// TIA Portal V18 export
FUNCTION "Boiler_UnitState" : Void   // FC61000, FBD
{ S7_Optimized_Access := 'TRUE' }
VERSION : 0.1
// BoilerOpMode                                        BoilerUnitState
// 0-OFF/Summer                                       0 Off
// 1-On/Winter                                             1 ColdStandBy
//                                                                   1 HotStandBy
//                                                                   2 Heating
// stored: AutoNumber false, IsIECCheckEnabled false, SetENOAutomatically false, UDAEnableTagReadback false
   VAR_INPUT
      rOAT : Real;
      rBoiler1OATOff : Real;
      rBoiler1OATOn : Real;
      rBoiler2OAT1On : Real;
      rBoiler2OAT1Off : Real;
      rBoiler2OAT2On : Real;
      rBoiler2OAT2Off : Real;
   END_VAR
   VAR_IN_OUT
      xBoiler1OATRequest : Bool;
      xBoiler2OATRequest : Bool;
   END_VAR
   VAR_TEMP
      FA_temp : Real;
      xB1State : Bool;
      xB2Band1State : Bool;
      xB2Band2State : Bool;
      xB2Band1Effective : Bool;
   END_VAR
BEGIN

REGION Network 1 (SCL)
   IF "FirstScan" THEN
       ;
       //"AHUUnitStates".UnitStates.cActual[#iUnitID] := 0;
       //"AHUUnitStates".UnitStates.cTarget[#iUnitID] := 0;
   END_IF;
END_REGION

REGION Network 2 (SCL): Boiler1 Select from Panel
   IF "HSsDI".Requests.xSeasonAuto[1] THEN
       "BoilerOpModes".OpModes.cPreselectedOpModePanel[1] := 2;//Auto
   ELSIF "HSsDI".Requests.xSeasonWinter[1] THEN
       "BoilerOpModes".OpModes.cPreselectedOpModePanel[1]:= 1;//Winter - Always On
   ELSE
       "BoilerOpModes".OpModes.cPreselectedOpModePanel[1] := 0;//Summer - Off
   END_IF;
END_REGION

REGION Network 3 (SCL): Boiler2 Select from Panel
   IF "BoilerOpModes".OpModes.xBoiler2IndividualPanelSwitch THEN
       IF "HSsDI".Requests.xSeasonAuto[2] THEN
           "BoilerOpModes".OpModes.cPreselectedOpModePanel[2] := 2;//Auto
       ELSIF "HSsDI".Requests.xSeasonWinter[2] THEN
           "BoilerOpModes".OpModes.cPreselectedOpModePanel[2] := 1;//Winter - Always On
       ELSE
           "BoilerOpModes".OpModes.cPreselectedOpModePanel[2] := 0;//Summer - Off
       END_IF;
   ELSE
       IF "HSsDI".Requests.xSeasonAuto[1] THEN
           "BoilerOpModes".OpModes.cPreselectedOpModePanel[2] := 2;//Auto
       ELSIF "HSsDI".Requests.xSeasonWinter[1] THEN
           "BoilerOpModes".OpModes.cPreselectedOpModePanel[2] := 1;//Winter - Always On
       ELSE
           "BoilerOpModes".OpModes.cPreselectedOpModePanel[2] := 0;//Summer - Off
       END_IF;
   END_IF;
END_REGION

REGION Network 4: Boiler1 Actual Operation Mode define
   // Operation Modes                                                 Unit State
   // 0=Protection                                                         0=Stopped
   // 1=Economy                                                           1=Checking-up  
   // 2=PreComfort                                                       2=Preheating
   // 3=Comfor                                                              3=Starting 
   // 4=Auto(Scheduler)                                              4=RecirculatingOperation (Protection)
   //                                                                                 5=Sustained Mode (Economy setpoints)
   //                                                                                 6=Sustained Mode (PreComfort setpoints) 
   //                                                                                 7=Comfort  operation
   //                                                                                 8=Stopping
   //                                                                                 9=Blocking
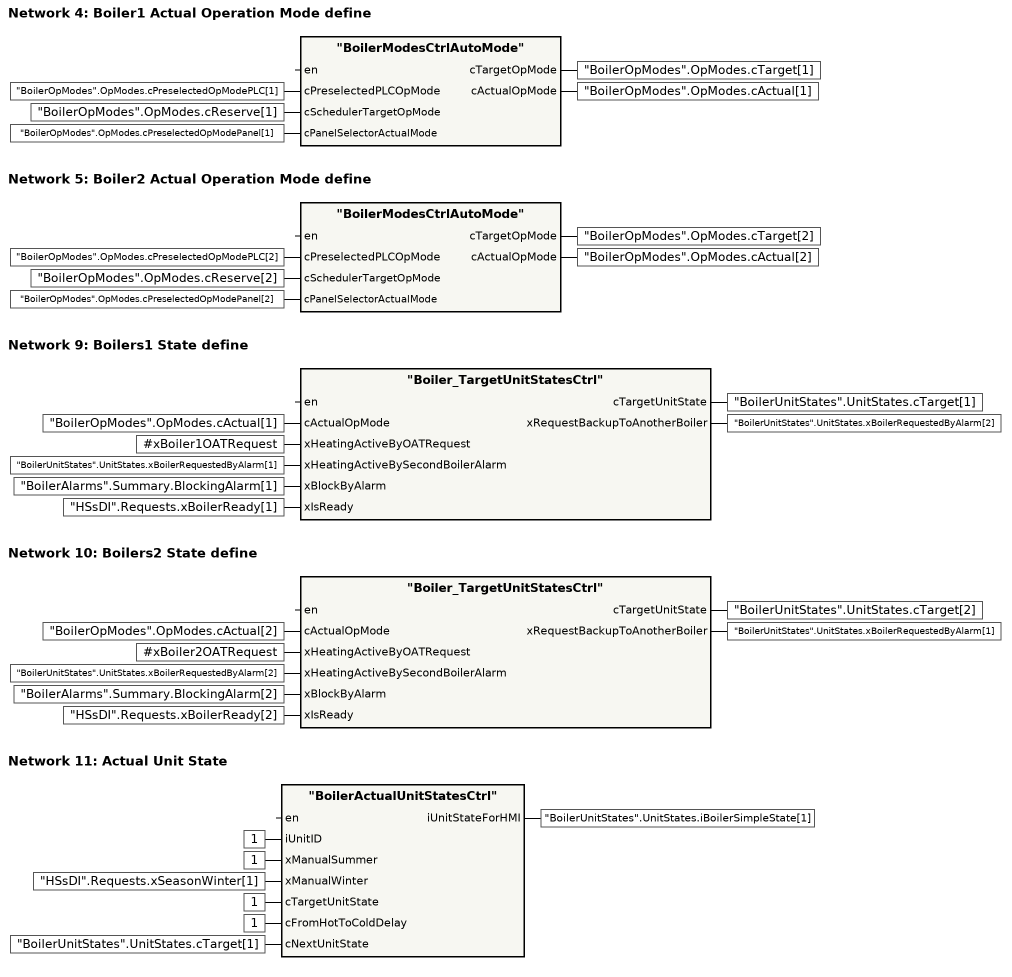
   "BoilerModesCtrlAutoMode"(cPreselectedPLCOpMode := "BoilerOpModes".OpModes.cPreselectedOpModePLC[1],
                           cSchedulerTargetOpMode := "BoilerOpModes".OpModes.cReserve[1],
                           cPanelSelectorActualMode := "BoilerOpModes".OpModes.cPreselectedOpModePanel[1],
                           cTargetOpMode => "BoilerOpModes".OpModes.cTarget[1],
                           cActualOpMode => "BoilerOpModes".OpModes.cActual[1]);
END_REGION

REGION Network 5: Boiler2 Actual Operation Mode define
   "BoilerModesCtrlAutoMode"(cPreselectedPLCOpMode := "BoilerOpModes".OpModes.cPreselectedOpModePLC[2],
                           cSchedulerTargetOpMode := "BoilerOpModes".OpModes.cReserve[2],
                           cPanelSelectorActualMode := "BoilerOpModes".OpModes.cPreselectedOpModePanel[2],
                           cTargetOpMode => "BoilerOpModes".OpModes.cTarget[2],
                           cActualOpMode => "BoilerOpModes".OpModes.cActual[2]);
END_REGION

REGION Network 6 (SCL): Boiler1 request by OAT
   IF NOT #xB1State THEN
       // Вмикаємо котел 1, коли стало достатньо холодно
       IF #rOAT <= #rBoiler1OATOn THEN
           #xB1State := TRUE;
       END_IF;
   ELSE
       // Вимикаємо котел 1, коли потеплішало вище абсолютного порогу
       IF #rOAT >= #rBoiler1OATOff THEN
           #xB1State := FALSE;
       END_IF;
   END_IF;

   #xBoiler1OATRequest := #xB1State;
END_REGION

REGION Network 7 (SCL): Boiler2 request by OAT, OAT range 1
   // Помірний холод»Помірний холод»: дозволяти лише доти, доки котел 1 ще НЕ увімкнувся.
   // // Пороги незалежні й реалізовані абсолютними значеннями
   IF NOT #xB2Band1State THEN
       IF #rOAT <= #rBoiler2OAT1On THEN
           #xB2Band1State := TRUE;
       END_IF;
   ELSE
       IF #rOAT >= #rBoiler2OAT1Off THEN
           #xB2Band1State := FALSE;
       END_IF;
   END_IF;

   // Маскуємо Band1, якщо котел 1 вже дозволений (умова "до включення першого котла")
   #xB2Band1Effective := #xB2Band1State AND (NOT #xBoiler1OATRequest);
END_REGION

REGION Network 8 (SCL): Boiler2 request by OAT, OAT range 2
   // «Сильний мороз»: дозволяти незалежно від стану котла 1.
   IF NOT #xB2Band2State THEN
       IF #rOAT <= #rBoiler2OAT2On THEN
           #xB2Band2State := TRUE;
       END_IF;
   ELSE
       IF #rOAT >= #rBoiler2OAT2Off THEN
           #xB2Band2State := FALSE;
       END_IF;
   END_IF;

   #xBoiler2OATRequest := #xB2Band2State OR #xB2Band1Effective;
END_REGION

REGION Network 9: Boilers1 State define
   // Operation Modes                                                 Unit State
   "Boiler_TargetUnitStatesCtrl"(cActualOpMode := "BoilerOpModes".OpModes.cActual[1],
                           xHeatingActiveByOATRequest := #xBoiler1OATRequest,
                           xHeatingActiveBySecondBoilerAlarm := "BoilerUnitStates".UnitStates.xBoilerRequestedByAlarm[1],
                           xBlockByAlarm := "BoilerAlarms".Summary.BlockingAlarm[1],
                           xIsReady := "HSsDI".Requests.xBoilerReady[1],
                           cTargetUnitState => "BoilerUnitStates".UnitStates.cTarget[1],
                           xRequestBackupToAnotherBoiler => "BoilerUnitStates".UnitStates.xBoilerRequestedByAlarm[2]);
END_REGION

REGION Network 10: Boilers2 State define
   // Operation Modes                                                 Unit State
   "Boiler_TargetUnitStatesCtrl"(cActualOpMode := "BoilerOpModes".OpModes.cActual[2],
                           xHeatingActiveByOATRequest := #xBoiler2OATRequest,
                           xHeatingActiveBySecondBoilerAlarm := "BoilerUnitStates".UnitStates.xBoilerRequestedByAlarm[2],
                           xBlockByAlarm := "BoilerAlarms".Summary.BlockingAlarm[2],
                           xIsReady := "HSsDI".Requests.xBoilerReady[2],
                           cTargetUnitState => "BoilerUnitStates".UnitStates.cTarget[2],
                           xRequestBackupToAnotherBoiler => "BoilerUnitStates".UnitStates.xBoilerRequestedByAlarm[1]);
END_REGION

REGION Network 11: Actual Unit State
   "BoilerActualUnitStatesCtrl"(iUnitID := 1,
                           xManualSummer := 1,
                           xManualWinter := "HSsDI".Requests.xSeasonWinter[1],
                           cTargetUnitState := 1,
                           cFromHotToColdDelay := 1,
                           cNextUnitState := "BoilerUnitStates".UnitStates.cTarget[1],
                           iUnitStateForHMI => "BoilerUnitStates".UnitStates.iBoilerSimpleState[1]);
END_REGION
END_FUNCTION
